(* PLC project CoDeSys External Library Template, WAGO e!COCKPIT e!COCKPIT, author 3S - Smart Software Solutions GmbH *)
(* stored: creationDateTime 2019-10-29T14:38:30.855626, version 3.5.5.30, modificationDateTime 2019-10-29T14:38:06.5373783, organization 3S - Smart Software Solutions GmbH *)
(* Library project template with all possible element types, docu and a sample project structure *)

FUNCTION_BLOCK fbPPPSAnalizatorDirisA40
  VAR_INPUT
    sKomunikat : alSTRINGKomunikat;  (* komunikat z systemu zewnętrznego *)
    intTablicaKomunikatowRozmiar : INT;  (* rozmiar tablicy danych wysyłkowych *)
    xTablicaKomunikatowHold : BOOL;  (* wstrzymanie komunikacji mniej ważnych komunikatów *)
    sIdInstancji : STRING;  (* parametr ID rolety np NS02L*202IBM**** *)
    sIdAplikacji : STRING;  (* parametr ID aplikacji np SO*******ECL*000 *)
    sMnemonik : STRING;  (* mnemonik właściciela - BCB* *)
    sMACAdres : STRING;  (* MAC adres sterownika *)
    sDaneZapasowe : STRING;  (* 6 znaków zapasu *)
    tCzasOpoznieniaRestartu : TIME;  (* czas opóźnienia po którym zaczynają być raportowane wartości *)
    bAdres : BYTE;
    rDeadband : REAL;
    tMinimalnyCzasRaportowania : TIME;
    tMaksymalnyCzasRaportowania : TIME;
    xAutonomizacja : BOOL;
  END_VAR
  VAR_IN_OUT
    arModbusOdczytCykliczny : ARRAY[1..5000] OF typModbusOdczytCykliczny;
    arModbusStatusKomunikacji : ARRAY[1..256] OF INT;
    arTablicaKomunikatow : alARRAYTablicaKomunikatow;
    intTablicaKomunikatowZnacznikZapisu : INT;
  END_VAR
  VAR
    xPierwszySkan : BOOL := TRUE;
    intPetlaPierwszySkan : INT := 1;
    fbTimerBrakuKomunikacji : TON;  (* Kontrola komunikacji urządzenia *)
    xBrakKomunikacjiPLC : BOOL;
    xBrakKomunikacjiIZE : BOOL;
    wNapiecieL1Hi : WORD;  (* Napięcia fazowe *)
    wNapiecieL1Lo : WORD;
    rNapiecieL1 : REAL;
    fbNapiecieL1 : fbFiltrWartoscAnalogowa;
    rNapiecieL1Zaraportowana : REAL;
    rNapiecieL1Pamiec : REAL;
    xBrakZmianyNapiecieL1 : BOOL;
    fbBrakZmianyNapiecieL1Timer : TON;
    xBladBrakZmianyNapiecieL1 : BOOL;
    wNapiecieL2Hi : WORD;
    wNapiecieL2Lo : WORD;
    rNapiecieL2 : REAL;
    fbNapiecieL2 : fbFiltrWartoscAnalogowa;
    rNapiecieL2Zaraportowana : REAL;
    rNapiecieL2Pamiec : REAL;
    xBrakZmianyNapiecieL2 : BOOL;
    fbBrakZmianyNapiecieL2Timer : TON;
    xBladBrakZmianyNapiecieL2 : BOOL;
    wNapiecieL3Hi : WORD;
    wNapiecieL3Lo : WORD;
    rNapiecieL3 : REAL;
    fbNapiecieL3 : fbFiltrWartoscAnalogowa;
    rNapiecieL3Zaraportowana : REAL;
    rNapiecieL3Pamiec : REAL;
    xBrakZmianyNapiecieL3 : BOOL;
    fbBrakZmianyNapiecieL3Timer : TON;
    xBladBrakZmianyNapiecieL3 : BOOL;
    wNapiecieL1L2Hi : WORD;  (* Napięcia przewodowe *)
    wNapiecieL1L2Lo : WORD;
    rNapiecieL1L2 : REAL;
    fbNapiecieL1L2 : fbFiltrWartoscAnalogowa;
    rNapiecieL1L2Zaraportowana : REAL;
    wNapiecieL2L3Hi : WORD;
    wNapiecieL2L3Lo : WORD;
    rNapiecieL2L3 : REAL;
    fbNapiecieL2L3 : fbFiltrWartoscAnalogowa;
    rNapiecieL2L3Zaraportowana : REAL;
    wNapiecieL3L1Hi : WORD;
    wNapiecieL3L1Lo : WORD;
    rNapiecieL3L1 : REAL;
    fbNapiecieL3L1 : fbFiltrWartoscAnalogowa;
    rNapiecieL3L1Zaraportowana : REAL;
    wCzestotliwoscHi : WORD;  (* Częstotliwość *)
    wCzestotliwoscLo : WORD;
    rCzestotliwosc : REAL;
    fbCzestotliwosc : fbFiltrWartoscAnalogowa;
    rCzestotliwoscZaraportowana : REAL;
    wCzasPracyAnalizatoraHi : WORD;  (* Czas pracy *)
    wCzasPracyAnalizatoraLo : WORD;
    rCzasPracyAnalizatora : REAL;
    fbCzasPracyAnalizatora : fbFiltrWartoscAnalogowa;
    rCzasPracyAnalizatoraZaraportowana : REAL;
    wPradL1Hi : WORD;  (* Prądy fazowe *)
    wPradL1Lo : WORD;
    rPradL1 : REAL;
    fbPradL1 : fbFiltrWartoscAnalogowa;
    rPradL1Zaraportowana : REAL;
    rPradL1Pamiec : REAL;
    xBrakZmianyPradL1 : BOOL;
    fbBrakZmianyPradL1Timer : TON;
    xBladBrakZmianyPradL1 : BOOL;
    wPradL2Hi : WORD;
    wPradL2Lo : WORD;
    rPradL2 : REAL;
    fbPradL2 : fbFiltrWartoscAnalogowa;
    rPradL2Zaraportowana : REAL;
    rPradL2Pamiec : REAL;
    xBrakZmianyPradL2 : BOOL;
    fbBrakZmianyPradL2Timer : TON;
    xBladBrakZmianyPradL2 : BOOL;
    wPradL3Hi : WORD;
    wPradL3Lo : WORD;
    rPradL3 : REAL;
    fbPradL3 : fbFiltrWartoscAnalogowa;
    rPradL3Zaraportowana : REAL;
    rPradL3Pamiec : REAL;
    xBrakZmianyPradL3 : BOOL;
    fbBrakZmianyPradL3Timer : TON;
    xBladBrakZmianyPradL3 : BOOL;
    wPradNHi : WORD;
    wPradNLo : WORD;
    rPradN : REAL;
    fbPradN : fbFiltrWartoscAnalogowa;
    rPradNZaraportowana : REAL;
    wPradSredniL1Hi : WORD;  (* Prądy średnie fazowe *)
    wPradSredniL1Lo : WORD;
    rPradSredniL1 : REAL;
    fbPradSredniL1 : fbFiltrWartoscAnalogowa;
    rPradSredniL1Zaraportowana : REAL;
    wPradSredniL2Hi : WORD;
    wPradSredniL2Lo : WORD;
    rPradSredniL2 : REAL;
    fbPradSredniL2 : fbFiltrWartoscAnalogowa;
    rPradSredniL2Zaraportowana : REAL;
    wPradSredniL3Hi : WORD;
    wPradSredniL3Lo : WORD;
    rPradSredniL3 : REAL;
    fbPradSredniL3 : fbFiltrWartoscAnalogowa;
    rPradSredniL3Zaraportowana : REAL;
    rPradSredni : REAL;  (* Prąd średni (I1+I2+I3)/3 *)
    fbPradSredni : fbFiltrWartoscAnalogowa;
    rPradSredniZaraportowana : REAL;
    wMocCzynnaCalkowitaHi : WORD;  (* Moc 3-fazowa czynna *)
    wMocCzynnaCalkowitaLo : WORD;
    rMocCzynnaCalkowita : REAL;
    fbMocCzynnaCalkowita : fbFiltrWartoscAnalogowa;
    rMocCzynnaCalkowitaZaraportowana : REAL;
    wMocBiernaCalkowitaHi : WORD;  (* Moc 3-fazowa bierna *)
    wMocBiernaCalkowitaLo : WORD;
    rMocBiernaCalkowita : REAL;
    fbMocBiernaCalkowita : fbFiltrWartoscAnalogowa;
    rMocBiernaCalkowitaZaraportowana : REAL;
    wMocPozornaCalkowitaHi : WORD;  (* Moc 3-fazowa pozorna *)
    wMocPozornaCalkowitaLo : WORD;
    rMocPozornaCalkowita : REAL;
    fbMocPozornaCalkowita : fbFiltrWartoscAnalogowa;
    rMocPozornaCalkowitaZaraportowana : REAL;
    wWspolczynnikMocyCalkowityHi : WORD;  (* Całkowity współczynnik mocy *)
    wWspolczynnikMocyCalkowityLo : WORD;
    rWspolczynnikMocyCalkowity : REAL;
    fbWspolczynnikMocyCalkowity : fbFiltrWartoscAnalogowa;
    rWspolczynnikMocyCalkowityZaraportowana : REAL;
    wMocCzynnaL1Hi : WORD;  (* Moc Czynna fazowa *)
    wMocCzynnaL1Lo : WORD;
    rMocCzynnaL1 : REAL;
    fbMocCzynnaL1 : fbFiltrWartoscAnalogowa;
    rMocCzynnaL1Zaraportowana : REAL;
    wMocCzynnaL2Hi : WORD;
    wMocCzynnaL2Lo : WORD;
    rMocCzynnaL2 : REAL;
    fbMocCzynnaL2 : fbFiltrWartoscAnalogowa;
    rMocCzynnaL2Zaraportowana : REAL;
    wMocCzynnaL3Hi : WORD;
    wMocCzynnaL3Lo : WORD;
    rMocCzynnaL3 : REAL;
    fbMocCzynnaL3 : fbFiltrWartoscAnalogowa;
    rMocCzynnaL3Zaraportowana : REAL;
    wMocBiernaL1Hi : WORD;  (* Moc Bierna fazowa *)
    wMocBiernaL1Lo : WORD;
    rMocBiernaL1 : REAL;
    fbMocBiernaL1 : fbFiltrWartoscAnalogowa;
    rMocBiernaL1Zaraportowana : REAL;
    wMocBiernaL2Hi : WORD;
    wMocBiernaL2Lo : WORD;
    rMocBiernaL2 : REAL;
    fbMocBiernaL2 : fbFiltrWartoscAnalogowa;
    rMocBiernaL2Zaraportowana : REAL;
    wMocBiernaL3Hi : WORD;
    wMocBiernaL3Lo : WORD;
    rMocBiernaL3 : REAL;
    fbMocBiernaL3 : fbFiltrWartoscAnalogowa;
    rMocBiernaL3Zaraportowana : REAL;
    wMocPozornaL1Hi : WORD;  (* Moc Pozorna fazowa *)
    wMocPozornaL1Lo : WORD;
    rMocPozornaL1 : REAL;
    fbMocPozornaL1 : fbFiltrWartoscAnalogowa;
    rMocPozornaL1Zaraportowana : REAL;
    wMocPozornaL2Hi : WORD;
    wMocPozornaL2Lo : WORD;
    rMocPozornaL2 : REAL;
    fbMocPozornaL2 : fbFiltrWartoscAnalogowa;
    rMocPozornaL2Zaraportowana : REAL;
    wMocPozornaL3Hi : WORD;
    wMocPozornaL3Lo : WORD;
    rMocPozornaL3 : REAL;
    fbMocPozornaL3 : fbFiltrWartoscAnalogowa;
    rMocPozornaL3Zaraportowana : REAL;
    wWspolczynnikMocyL1Hi : WORD;  (* Fazowe współczynniki mocy *)
    wWspolczynnikMocyL1Lo : WORD;
    rWspolczynnikMocyL1 : REAL;
    fbWspolczynnikMocyL1 : fbFiltrWartoscAnalogowa;
    rWspolczynnikMocyL1Zaraportowana : REAL;
    wWspolczynnikMocyL2Hi : WORD;
    wWspolczynnikMocyL2Lo : WORD;
    rWspolczynnikMocyL2 : REAL;
    fbWspolczynnikMocyL2 : fbFiltrWartoscAnalogowa;
    rWspolczynnikMocyL2Zaraportowana : REAL;
    wWspolczynnikMocyL3Hi : WORD;
    wWspolczynnikMocyL3Lo : WORD;
    rWspolczynnikMocyL3 : REAL;
    fbWspolczynnikMocyL3 : fbFiltrWartoscAnalogowa;
    rWspolczynnikMocyL3Zaraportowana : REAL;
    wEnergiaCzynnaPobranaHi : WORD;  (* Energia pobrana *)
    wEnergiaCzynnaPobranaLo : WORD;
    rEnergiaCzynnaPobrana : REAL;
    fbEnergiaCzynnaPobrana : fbFiltrWartoscAnalogowa;
    rEnergiaCzynnaPobranaZaraportowana : REAL;
    wEnergiaBiernaPobranaHi : WORD;
    wEnergiaBiernaPobranaLo : WORD;
    rEnergiaBiernaPobrana : REAL;
    fbEnergiaBiernaPobrana : fbFiltrWartoscAnalogowa;
    rEnergiaBiernaPobranaZaraportowana : REAL;
    wEnergiaPozornaPobranaHi : WORD;
    wEnergiaPozornaPobranaLo : WORD;
    rEnergiaPozornaPobrana : REAL;
    fbEnergiaPozornaPobrana : fbFiltrWartoscAnalogowa;
    rEnergiaPozornaPobranaZaraportowana : REAL;
    wMocCzynnaSredniaHi : WORD;  (* Moc średnia *)
    wMocCzynnaSredniaLo : WORD;
    rMocCzynnaSrednia : REAL;
    fbMocCzynnaSrednia : fbFiltrWartoscAnalogowa;
    rMocCzynnaSredniaZaraportowana : REAL;
    wMocBiernaSredniaHi : WORD;
    wMocBiernaSredniaLo : WORD;
    rMocBiernaSrednia : REAL;
    fbMocBiernaSrednia : fbFiltrWartoscAnalogowa;
    rMocBiernaSredniaZaraportowana : REAL;
    wMocPozornaSredniaHi : WORD;
    wMocPozornaSredniaLo : WORD;
    rMocPozornaSrednia : REAL;
    fbMocPozornaSrednia : fbFiltrWartoscAnalogowa;
    rMocPozornaSredniaZaraportowana : REAL;
    wMaksymalneNapiecieL1Hi : WORD;  (* Maksymalne napięcia fazowe *)
    wMaksymalneNapiecieL1Lo : WORD;
    rMaksymalneNapiecieL1 : REAL;
    fbMaksymalneNapiecieL1 : fbFiltrWartoscAnalogowa;
    rMaksymalneNapiecieL1Zaraportowana : REAL;
    wMaksymalneNapiecieL2Hi : WORD;
    wMaksymalneNapiecieL2Lo : WORD;
    rMaksymalneNapiecieL2 : REAL;
    fbMaksymalneNapiecieL2 : fbFiltrWartoscAnalogowa;
    rMaksymalneNapiecieL2Zaraportowana : REAL;
    wMaksymalneNapiecieL3Hi : WORD;
    wMaksymalneNapiecieL3Lo : WORD;
    rMaksymalneNapiecieL3 : REAL;
    fbMaksymalneNapiecieL3 : fbFiltrWartoscAnalogowa;
    rMaksymalneNapiecieL3Zaraportowana : REAL;
    wTHDNapieciaL1 : WORD;  (* THD napięcia *)
    rTHDNapieciaL1 : REAL;
    fbTHDNapieciaL1 : fbFiltrWartoscAnalogowa;
    rTHDNapieciaL1Zaraportowana : REAL;
    wTHDNapieciaL2 : WORD;
    rTHDNapieciaL2 : REAL;
    fbTHDNapieciaL2 : fbFiltrWartoscAnalogowa;
    rTHDNapieciaL2Zaraportowana : REAL;
    wTHDNapieciaL3 : WORD;
    rTHDNapieciaL3 : REAL;
    fbTHDNapieciaL3 : fbFiltrWartoscAnalogowa;
    rTHDNapieciaL3Zaraportowana : REAL;
    wTHDPraduL1 : WORD;  (* THD prądu *)
    rTHDPraduL1 : REAL;
    fbTHDPraduL1 : fbFiltrWartoscAnalogowa;
    rTHDPraduL1Zaraportowana : REAL;
    wTHDPraduL2 : WORD;
    rTHDPraduL2 : REAL;
    fbTHDPraduL2 : fbFiltrWartoscAnalogowa;
    rTHDPraduL2Zaraportowana : REAL;
    wTHDPraduL3 : WORD;
    rTHDPraduL3 : REAL;
    fbTHDPraduL3 : fbFiltrWartoscAnalogowa;
    rTHDPraduL3Zaraportowana : REAL;
    xPoInicjalizacji : BOOL;  (* inicjalizacja *)
    fbInicjalizacyjnyTimer : TON;
    intStatus : INT := enumPPPSUrzadenieStatus.Prawidlowy;  (* status urządzenia *)
    intStatusZaraportowana : INT;  (* status urządzenia zaraportowany *)
    sDane : alSTRINGKomunikat;
    sWyslanyKomunikat : alSTRINGKomunikat;
    xZadanieRaportu : BOOL;
    sWyslanyKomunikatDummy : alSTRINGKomunikat;
    sKomunikatPamiec : alSTRINGKomunikat;
    intPetla : INT;
    arErrorStan : ARRAY[0..20] OF INT;  (* tablica przechowująca statusy alarmowe *)
    arErrorKlasa : ARRAY[0..20] OF INT;  (* tablica przechowująca klasy danych alarmów *)
    xRaport : BOOL := FALSE;
    xOverFlow : BOOL;
  END_VAR

            (*			
Autor:					Paweł Kąkol, 2018-09-04-PK
Prawa majątkowe: 		Solwena Sp. z o.o., 
Opis:					fb służy do komunikacji po Modbus RTU z analizatorem sieci ECA0 na budynkach PPP Sopot
						Analizator Diris A40
						
Aktualizacje:			2018-11-20-JB: Poprawienie adresów Modbusowych
						2019-01-21-JC: Przeliczanie charakteru mocy biernej oraz współczynnika mocy (czynna/indukcyjna)
						2019-03-26-AWy: Wyłączenie (wykomentowanie) eneregii oddanej czynnej i biernej
						2019-04-01-AWy: Przeliczenie pomocnicze dla mocy czynnej całkowitej
						2019-05-05-AWy: Dodanie bloków włączania autonomizacji i kontroli komunikacji (analogicznie do pozostałych fb). Usunięcie zmiennej xBrakKomunikacji
						2019-08-14-AWy: Przeniesienie xAutonomizacja do VAR_INPUT
						2019-09-04-AWy: Usunięcie bugów z obliczania współczynnika mocy i mocy biernej.
						2019-09-05-Awy: Zmiana sposobu przeliczania wartości odczytanych po modbusie (sklejenie w DINT i konwersja na REAL). Usunięcie energii oddanej czynnej i biernej.
										Zmiana nazwy atrybutu FACTOR na FACTOR3PH.
						2019-10-18-JB: Zmiana dead-bandów.
						2019-10-24-AWy: Zmiana wartości tCzasMinimalny dla czasu pracy analizatora.
	
*)

//inicjalizacja sterownika

fbInicjalizacyjnyTimer(IN := NOT xPoInicjalizacji , PT := tCzasOpoznieniaRestartu);
IF fbInicjalizacyjnyTimer.Q THEN
	rNapiecieL1Zaraportowana := rNapiecieL1;
	rNapiecieL2Zaraportowana := rNapiecieL2;
	rNapiecieL3Zaraportowana :=sdfsdgsdf rNapiecieL3;
	rNapiecieL1L2Zaraportowana := rNapiecieL1L2;
	rNapiecieL2L3Zaraportowana := rNapiecieL2L3;
	rNapiecieL3L1Zaraportowana := rNapiecieL3L1;
	rCzestotliwoscZaraportowana := rCzestotliwosc;
	rCzasPracyAnalizatoraZaraportowana := rCzasPracyAnalizatora;
	rPradL1Zaraportowana := rPradL1;
	rPradL2Zaraportowana := rPradL2;
	rPradL3Zaraportowana := rPradL3;
	rPradNZaraportowana := rPradN;
	rPradSredniL1Zaraportowana := rPradSredniL1;
	rPradSredniL2Zaraportowana := rPradSredniL2;
	rPradSredniL3Zaraportowana := rPradSredniL3;
	rPradSredniZaraportowana := rPradSredni;
	rMocCzynnaCalkowitaZaraportowana := rMocCzynnaCalkowita;
	rMocBiernaCalkowitaZaraportowana := rMocBiernaCalkowita;
	rMocPozornaCalkowitaZaraportowana := rMocPozornaCalkowita;
	rWspolczynnikMocyCalkowityZaraportowana := rWspolczynnikMocyCalkowity;
	rMocCzynnaL1Zaraportowana := rMocCzynnaL1;
	rMocCzynnaL2Zaraportowana := rMocCzynnaL2;
	rMocCzynnaL3Zaraportowana := rMocCzynnaL3;
	rMocBiernaL1Zaraportowana := rMocBiernaL1;
	rMocBiernaL2Zaraportowana := rMocBiernaL2;
	rMocBiernaL3Zaraportowana := rMocBiernaL3;
	rMocPozornaL1Zaraportowana := rMocPozornaL1;
	rMocPozornaL2Zaraportowana := rMocPozornaL2;
	rMocPozornaL3Zaraportowana := rMocPozornaL3;
	rWspolczynnikMocyL1Zaraportowana := rWspolczynnikMocyL1;
	rWspolczynnikMocyL2Zaraportowana := rWspolczynnikMocyL2;
	rWspolczynnikMocyL3Zaraportowana := rWspolczynnikMocyL3;
	rEnergiaCzynnaPobranaZaraportowana := rEnergiaCzynnaPobrana;
	rEnergiaBiernaPobranaZaraportowana := rEnergiaBiernaPobrana;
	rEnergiaPozornaPobranaZaraportowana := rEnergiaPozornaPobrana;
	rMocCzynnaSredniaZaraportowana := rMocCzynnaSrednia;
	rMocBiernaSredniaZaraportowana := rMocBiernaSrednia;
	rMocPozornaSredniaZaraportowana := rMocPozornaSrednia;
	rMaksymalneNapiecieL1Zaraportowana := rMaksymalneNapiecieL1;
	rMaksymalneNapiecieL2Zaraportowana := rMaksymalneNapiecieL2;
	rMaksymalneNapiecieL3Zaraportowana := rMaksymalneNapiecieL3;
	rTHDNapieciaL1Zaraportowana := rTHDNapieciaL1;
	rTHDNapieciaL2Zaraportowana := rTHDNapieciaL2;
	rTHDNapieciaL3Zaraportowana := rTHDNapieciaL3;
	rTHDPraduL1Zaraportowana := rTHDPraduL1;
	rTHDPraduL2Zaraportowana := rTHDPraduL2;
	rTHDPraduL3Zaraportowana := rTHDPraduL3;
	intStatusZaraportowana := intStatus;
	xPoInicjalizacji := TRUE;
	dupa dupa dupa
END_IF

// Włącz autonomizację jeśli sterownik jest w stanie inicjalizacji lub nastąpiło wymuszenie autonomizacji
IF NOT xPoInicjalizacji THEN
	xAutonomizacja := TRUE;
END_IF 

// Kontrola komunikacji
fbTimerBrakuKomunikacji(IN := arModbusStatusKomunikacji[bAdres] = enumModbusStatus.BrakKomunikacji, PT := T#60S);
IF fbTimerBrakuKomunikacji.Q THEN
	xBrakKomunikacjiPLC := TRUE;
ELSE
	xBrakKomunikacjiPLC := FALSE;
END_IF

IF xAutonomizacja THEN
	xBrakKomunikacjiIZE := TRUE;
ELSE
	xBrakKomunikacjiIZE := FALSE;
END_IF

IF xPierwszySkan THEN
	xPierwszySkan := FALSE;
	WHILE arModbusOdczytCykliczny[intPetlaPierwszySkan].bAdresUrzadzenia <> 0 DO
		intPetlaPierwszySkan := intPetlaPierwszySkan + 1;
	END_WHILE

//deklaracja rejestrow do odczytu
	arModbusOdczytCykliczny[intPetlaPierwszySkan].bAdresUrzadzenia := bAdres;
	arModbusOdczytCykliczny[intPetlaPierwszySkan].bFunkcja := TO_BYTE(enumModbusKodyFunkcji.OdczytNRejestrow);
	arModbusOdczytCykliczny[intPetlaPierwszySkan].uiAdresRejestru := 50512;
	arModbusOdczytCykliczny[intPetlaPierwszySkan].ltCzestotliwosc := TIME_TO_LTIME(tMaksymalnyCzasRaportowania);
	arModbusOdczytCykliczny[intPetlaPierwszySkan].pZmiennaReferencyjna := ADR(wCzasPracyAnalizatoraHi);
	intPetlaPierwszySkan := intPetlaPierwszySkan + 1;

	arModbusOdczytCykliczny[intPetlaPierwszySkan].bAdresUrzadzenia := bAdres;
	arModbusOdczytCykliczny[intPetlaPierwszySkan].bFunkcja := TO_BYTE(enumModbusKodyFunkcji.OdczytNRejestrow);
	arModbusOdczytCykliczny[intPetlaPierwszySkan].uiAdresRejestru := 50513;
	arModbusOdczytCykliczny[intPetlaPierwszySkan].ltCzestotliwosc := TIME_TO_LTIME(tMaksymalnyCzasRaportowania);
	arModbusOdczytCykliczny[intPetlaPierwszySkan].pZmiennaReferencyjna := ADR(wCzasPracyAnalizatoraLo);
	intPetlaPierwszySkan := intPetlaPierwszySkan + 1;

	arModbusOdczytCykliczny[intPetlaPierwszySkan].bAdresUrzadzenia := bAdres;
	arModbusOdczytCykliczny[intPetlaPierwszySkan].bFunkcja := TO_BYTE(enumModbusKodyFunkcji.OdczytNRejestrow);
	arModbusOdczytCykliczny[intPetlaPierwszySkan].uiAdresRejestru := 50514;
	arModbusOdczytCykliczny[intPetlaPierwszySkan].ltCzestotliwosc := TIME_TO_LTIME(tMinimalnyCzasRaportowania);
	arModbusOdczytCykliczny[intPetlaPierwszySkan].pZmiennaReferencyjna := ADR(wNapiecieL1L2Hi);
	intPetlaPierwszySkan := intPetlaPierwszySkan + 1;

	arModbusOdczytCykliczny[intPetlaPierwszySkan].bAdresUrzadzenia := bAdres;
	arModbusOdczytCykliczny[intPetlaPierwszySkan].bFunkcja := TO_BYTE(enumModbusKodyFunkcji.OdczytNRejestrow);
	arModbusOdczytCykliczny[intPetlaPierwszySkan].uiAdresRejestru := 50515;
	arModbusOdczytCykliczny[intPetlaPierwszySkan].ltCzestotliwosc := TIME_TO_LTIME(tMinimalnyCzasRaportowania);
	arModbusOdczytCykliczny[intPetlaPierwszySkan].pZmiennaReferencyjna := ADR(wNapiecieL1L2Lo);
	intPetlaPierwszySkan := intPetlaPierwszySkan + 1;

	arModbusOdczytCykliczny[intPetlaPierwszySkan].bAdresUrzadzenia := bAdres;
	arModbusOdczytCykliczny[intPetlaPierwszySkan].bFunkcja := TO_BYTE(enumModbusKodyFunkcji.OdczytNRejestrow);
	arModbusOdczytCykliczny[intPetlaPierwszySkan].uiAdresRejestru := 50516;
	arModbusOdczytCykliczny[intPetlaPierwszySkan].ltCzestotliwosc := TIME_TO_LTIME(tMinimalnyCzasRaportowania);
	arModbusOdczytCykliczny[intPetlaPierwszySkan].pZmiennaReferencyjna := ADR(wNapiecieL2L3Hi);
	intPetlaPierwszySkan := intPetlaPierwszySkan + 1;
	
	arModbusOdczytCykliczny[intPetlaPierwszySkan].bAdresUrzadzenia := bAdres;
	arModbusOdczytCykliczny[intPetlaPierwszySkan].bFunkcja := TO_BYTE(enumModbusKodyFunkcji.OdczytNRejestrow);
	arModbusOdczytCykliczny[intPetlaPierwszySkan].uiAdresRejestru := 50517;
	arModbusOdczytCykliczny[intPetlaPierwszySkan].ltCzestotliwosc := TIME_TO_LTIME(tMinimalnyCzasRaportowania);
	arModbusOdczytCykliczny[intPetlaPierwszySkan].pZmiennaReferencyjna := ADR(wNapiecieL2L3Lo);
	intPetlaPierwszySkan := intPetlaPierwszySkan + 1;

	arModbusOdczytCykliczny[intPetlaPierwszySkan].bAdresUrzadzenia := bAdres;
	arModbusOdczytCykliczny[intPetlaPierwszySkan].bFunkcja := TO_BYTE(enumModbusKodyFunkcji.OdczytNRejestrow);
	arModbusOdczytCykliczny[intPetlaPierwszySkan].uiAdresRejestru := 50518;
	arModbusOdczytCykliczny[intPetlaPierwszySkan].ltCzestotliwosc := TIME_TO_LTIME(tMinimalnyCzasRaportowania);
	arModbusOdczytCykliczny[intPetlaPierwszySkan].pZmiennaReferencyjna := ADR(wNapiecieL3L1Hi);
	intPetlaPierwszySkan := intPetlaPierwszySkan + 1;
	
	arModbusOdczytCykliczny[intPetlaPierwszySkan].bAdresUrzadzenia := bAdres;
	arModbusOdczytCykliczny[intPetlaPierwszySkan].bFunkcja := TO_BYTE(enumModbusKodyFunkcji.OdczytNRejestrow);
	arModbusOdczytCykliczny[intPetlaPierwszySkan].uiAdresRejestru := 50519;
	arModbusOdczytCykliczny[intPetlaPierwszySkan].ltCzestotliwosc := TIME_TO_LTIME(tMinimalnyCzasRaportowania);
	arModbusOdczytCykliczny[intPetlaPierwszySkan].pZmiennaReferencyjna := ADR(wNapiecieL3L1Lo);
	intPetlaPierwszySkan := intPetlaPierwszySkan + 1;

	arModbusOdczytCykliczny[intPetlaPierwszySkan].bAdresUrzadzenia := bAdres;
	arModbusOdczytCykliczny[intPetlaPierwszySkan].bFunkcja := TO_BYTE(enumModbusKodyFunkcji.OdczytNRejestrow);
	arModbusOdczytCykliczny[intPetlaPierwszySkan].uiAdresRejestru := 50520;
	arModbusOdczytCykliczny[intPetlaPierwszySkan].ltCzestotliwosc := TIME_TO_LTIME(tMinimalnyCzasRaportowania);
	arModbusOdczytCykliczny[intPetlaPierwszySkan].pZmiennaReferencyjna := ADR(wNapiecieL1Hi);
	intPetlaPierwszySkan := intPetlaPierwszySkan + 1;

	arModbusOdczytCykliczny[intPetlaPierwszySkan].bAdresUrzadzenia := bAdres;
	arModbusOdczytCykliczny[intPetlaPierwszySkan].bFunkcja := TO_BYTE(enumModbusKodyFunkcji.OdczytNRejestrow);
	arModbusOdczytCykliczny[intPetlaPierwszySkan].uiAdresRejestru := 50521;
	arModbusOdczytCykliczny[intPetlaPierwszySkan].ltCzestotliwosc := TIME_TO_LTIME(tMinimalnyCzasRaportowania);
	arModbusOdczytCykliczny[intPetlaPierwszySkan].pZmiennaReferencyjna := ADR(wNapiecieL1Lo);
	intPetlaPierwszySkan := intPetlaPierwszySkan + 1;

	arModbusOdczytCykliczny[intPetlaPierwszySkan].bAdresUrzadzenia := bAdres;
	arModbusOdczytCykliczny[intPetlaPierwszySkan].bFunkcja := TO_BYTE(enumModbusKodyFunkcji.OdczytNRejestrow);
	arModbusOdczytCykliczny[intPetlaPierwszySkan].uiAdresRejestru := 50522;
	arModbusOdczytCykliczny[intPetlaPierwszySkan].ltCzestotliwosc := TIME_TO_LTIME(tMinimalnyCzasRaportowania);
	arModbusOdczytCykliczny[intPetlaPierwszySkan].pZmiennaReferencyjna := ADR(wNapiecieL2Hi);
	intPetlaPierwszySkan := intPetlaPierwszySkan + 1;
	
	arModbusOdczytCykliczny[intPetlaPierwszySkan].bAdresUrzadzenia := bAdres;
	arModbusOdczytCykliczny[intPetlaPierwszySkan].bFunkcja := TO_BYTE(enumModbusKodyFunkcji.OdczytNRejestrow);
	arModbusOdczytCykliczny[intPetlaPierwszySkan].uiAdresRejestru := 50523;
	arModbusOdczytCykliczny[intPetlaPierwszySkan].ltCzestotliwosc := TIME_TO_LTIME(tMinimalnyCzasRaportowania);
	arModbusOdczytCykliczny[intPetlaPierwszySkan].pZmiennaReferencyjna := ADR(wNapiecieL2Lo);
	intPetlaPierwszySkan := intPetlaPierwszySkan + 1;

	arModbusOdczytCykliczny[intPetlaPierwszySkan].bAdresUrzadzenia := bAdres;
	arModbusOdczytCykliczny[intPetlaPierwszySkan].bFunkcja := TO_BYTE(enumModbusKodyFunkcji.OdczytNRejestrow);
	arModbusOdczytCykliczny[intPetlaPierwszySkan].uiAdresRejestru := 50524;
	arModbusOdczytCykliczny[intPetlaPierwszySkan].ltCzestotliwosc := TIME_TO_LTIME(tMinimalnyCzasRaportowania);
	arModbusOdczytCykliczny[intPetlaPierwszySkan].pZmiennaReferencyjna := ADR(wNapiecieL3Hi);
	intPetlaPierwszySkan := intPetlaPierwszySkan + 1;
	
	arModbusOdczytCykliczny[intPetlaPierwszySkan].bAdresUrzadzenia := bAdres;
	arModbusOdczytCykliczny[intPetlaPierwszySkan].bFunkcja := TO_BYTE(enumModbusKodyFunkcji.OdczytNRejestrow);
	arModbusOdczytCykliczny[intPetlaPierwszySkan].uiAdresRejestru := 50525;
	arModbusOdczytCykliczny[intPetlaPierwszySkan].ltCzestotliwosc := TIME_TO_LTIME(tMinimalnyCzasRaportowania);
	arModbusOdczytCykliczny[intPetlaPierwszySkan].pZmiennaReferencyjna := ADR(wNapiecieL3Lo);
	intPetlaPierwszySkan := intPetlaPierwszySkan + 1;

	arModbusOdczytCykliczny[intPetlaPierwszySkan].bAdresUrzadzenia := bAdres;
	arModbusOdczytCykliczny[intPetlaPierwszySkan].bFunkcja := TO_BYTE(enumModbusKodyFunkcji.OdczytNRejestrow);
	arModbusOdczytCykliczny[intPetlaPierwszySkan].uiAdresRejestru := 50526;
	arModbusOdczytCykliczny[intPetlaPierwszySkan].ltCzestotliwosc := TIME_TO_LTIME(tMinimalnyCzasRaportowania);
	arModbusOdczytCykliczny[intPetlaPierwszySkan].pZmiennaReferencyjna := ADR(wCzestotliwoscHi);
	intPetlaPierwszySkan := intPetlaPierwszySkan + 1;

	arModbusOdczytCykliczny[intPetlaPierwszySkan].bAdresUrzadzenia := bAdres;
	arModbusOdczytCykliczny[intPetlaPierwszySkan].bFunkcja := TO_BYTE(enumModbusKodyFunkcji.OdczytNRejestrow);
	arModbusOdczytCykliczny[intPetlaPierwszySkan].uiAdresRejestru := 50527;
	arModbusOdczytCykliczny[intPetlaPierwszySkan].ltCzestotliwosc := TIME_TO_LTIME(tMinimalnyCzasRaportowania);
	arModbusOdczytCykliczny[intPetlaPierwszySkan].pZmiennaReferencyjna := ADR(wCzestotliwoscLo);
	intPetlaPierwszySkan := intPetlaPierwszySkan + 1;

	arModbusOdczytCykliczny[intPetlaPierwszySkan].bAdresUrzadzenia := bAdres;
	arModbusOdczytCykliczny[intPetlaPierwszySkan].bFunkcja := TO_BYTE(enumModbusKodyFunkcji.OdczytNRejestrow);
	arModbusOdczytCykliczny[intPetlaPierwszySkan].uiAdresRejestru := 50528;
	arModbusOdczytCykliczny[intPetlaPierwszySkan].ltCzestotliwosc := TIME_TO_LTIME(tMinimalnyCzasRaportowania);
	arModbusOdczytCykliczny[intPetlaPierwszySkan].pZmiennaReferencyjna := ADR(wPradL1Hi);
	intPetlaPierwszySkan := intPetlaPierwszySkan + 1;

	arModbusOdczytCykliczny[intPetlaPierwszySkan].bAdresUrzadzenia := bAdres;
	arModbusOdczytCykliczny[intPetlaPierwszySkan].bFunkcja := TO_BYTE(enumModbusKodyFunkcji.OdczytNRejestrow);
	arModbusOdczytCykliczny[intPetlaPierwszySkan].uiAdresRejestru := 50529;
	arModbusOdczytCykliczny[intPetlaPierwszySkan].ltCzestotliwosc := TIME_TO_LTIME(tMinimalnyCzasRaportowania);
	arModbusOdczytCykliczny[intPetlaPierwszySkan].pZmiennaReferencyjna := ADR(wPradL1Lo);
	intPetlaPierwszySkan := intPetlaPierwszySkan + 1;

	arModbusOdczytCykliczny[intPetlaPierwszySkan].bAdresUrzadzenia := bAdres;
	arModbusOdczytCykliczny[intPetlaPierwszySkan].bFunkcja := TO_BYTE(enumModbusKodyFunkcji.OdczytNRejestrow);
	arModbusOdczytCykliczny[intPetlaPierwszySkan].uiAdresRejestru := 50530;
	arModbusOdczytCykliczny[intPetlaPierwszySkan].ltCzestotliwosc := TIME_TO_LTIME(tMinimalnyCzasRaportowania);
	arModbusOdczytCykliczny[intPetlaPierwszySkan].pZmiennaReferencyjna := ADR(wPradL2Hi);
	intPetlaPierwszySkan := intPetlaPierwszySkan + 1;

	arModbusOdczytCykliczny[intPetlaPierwszySkan].bAdresUrzadzenia := bAdres;
	arModbusOdczytCykliczny[intPetlaPierwszySkan].bFunkcja := TO_BYTE(enumModbusKodyFunkcji.OdczytNRejestrow);
	arModbusOdczytCykliczny[intPetlaPierwszySkan].uiAdresRejestru := 50531;
	arModbusOdczytCykliczny[intPetlaPierwszySkan].ltCzestotliwosc := TIME_TO_LTIME(tMinimalnyCzasRaportowania);
	arModbusOdczytCykliczny[intPetlaPierwszySkan].pZmiennaReferencyjna := ADR(wPradL2Lo);
	intPetlaPierwszySkan := intPetlaPierwszySkan + 1;

	arModbusOdczytCykliczny[intPetlaPierwszySkan].bAdresUrzadzenia := bAdres;
	arModbusOdczytCykliczny[intPetlaPierwszySkan].bFunkcja := TO_BYTE(enumModbusKodyFunkcji.OdczytNRejestrow);
	arModbusOdczytCykliczny[intPetlaPierwszySkan].uiAdresRejestru := 50532;
	arModbusOdczytCykliczny[intPetlaPierwszySkan].ltCzestotliwosc := TIME_TO_LTIME(tMinimalnyCzasRaportowania);
	arModbusOdczytCykliczny[intPetlaPierwszySkan].pZmiennaReferencyjna := ADR(wPradL3Hi);
	intPetlaPierwszySkan := intPetlaPierwszySkan + 1;

	arModbusOdczytCykliczny[intPetlaPierwszySkan].bAdresUrzadzenia := bAdres;
	arModbusOdczytCykliczny[intPetlaPierwszySkan].bFunkcja := TO_BYTE(enumModbusKodyFunkcji.OdczytNRejestrow);
	arModbusOdczytCykliczny[intPetlaPierwszySkan].uiAdresRejestru := 50533;
	arModbusOdczytCykliczny[intPetlaPierwszySkan].ltCzestotliwosc := TIME_TO_LTIME(tMinimalnyCzasRaportowania);
	arModbusOdczytCykliczny[intPetlaPierwszySkan].pZmiennaReferencyjna := ADR(wPradL3Lo);
	intPetlaPierwszySkan := intPetlaPierwszySkan + 1;

	arModbusOdczytCykliczny[intPetlaPierwszySkan].bAdresUrzadzenia := bAdres;
	arModbusOdczytCykliczny[intPetlaPierwszySkan].bFunkcja := TO_BYTE(enumModbusKodyFunkcji.OdczytNRejestrow);
	arModbusOdczytCykliczny[intPetlaPierwszySkan].uiAdresRejestru := 50534;
	arModbusOdczytCykliczny[intPetlaPierwszySkan].ltCzestotliwosc := TIME_TO_LTIME(tMinimalnyCzasRaportowania);
	arModbusOdczytCykliczny[intPetlaPierwszySkan].pZmiennaReferencyjna := ADR(wPradNHi);
	intPetlaPierwszySkan := intPetlaPierwszySkan + 1;

	arModbusOdczytCykliczny[intPetlaPierwszySkan].bAdresUrzadzenia := bAdres;
	arModbusOdczytCykliczny[intPetlaPierwszySkan].bFunkcja := TO_BYTE(enumModbusKodyFunkcji.OdczytNRejestrow);
	arModbusOdczytCykliczny[intPetlaPierwszySkan].uiAdresRejestru := 50535;
	arModbusOdczytCykliczny[intPetlaPierwszySkan].ltCzestotliwosc := TIME_TO_LTIME(tMinimalnyCzasRaportowania);
	arModbusOdczytCykliczny[intPetlaPierwszySkan].pZmiennaReferencyjna := ADR(wPradNLo);
	intPetlaPierwszySkan := intPetlaPierwszySkan + 1;
	
	arModbusOdczytCykliczny[intPetlaPierwszySkan].bAdresUrzadzenia := bAdres;
	arModbusOdczytCykliczny[intPetlaPierwszySkan].bFunkcja := TO_BYTE(enumModbusKodyFunkcji.OdczytNRejestrow);
	arModbusOdczytCykliczny[intPetlaPierwszySkan].uiAdresRejestru := 50536;
	arModbusOdczytCykliczny[intPetlaPierwszySkan].ltCzestotliwosc := TIME_TO_LTIME(tMinimalnyCzasRaportowania);
	arModbusOdczytCykliczny[intPetlaPierwszySkan].pZmiennaReferencyjna := ADR(wMocCzynnaCalkowitaHi);
	intPetlaPierwszySkan := intPetlaPierwszySkan + 1;
	
	arModbusOdczytCykliczny[intPetlaPierwszySkan].bAdresUrzadzenia := bAdres;
	arModbusOdczytCykliczny[intPetlaPierwszySkan].bFunkcja := TO_BYTE(enumModbusKodyFunkcji.OdczytNRejestrow);
	arModbusOdczytCykliczny[intPetlaPierwszySkan].uiAdresRejestru := 50537;
	arModbusOdczytCykliczny[intPetlaPierwszySkan].ltCzestotliwosc := TIME_TO_LTIME(tMinimalnyCzasRaportowania);
	arModbusOdczytCykliczny[intPetlaPierwszySkan].pZmiennaReferencyjna := ADR(wMocCzynnaCalkowitaLo);
	intPetlaPierwszySkan := intPetlaPierwszySkan + 1;
	
	arModbusOdczytCykliczny[intPetlaPierwszySkan].bAdresUrzadzenia := bAdres;
	arModbusOdczytCykliczny[intPetlaPierwszySkan].bFunkcja := TO_BYTE(enumModbusKodyFunkcji.OdczytNRejestrow);
	arModbusOdczytCykliczny[intPetlaPierwszySkan].uiAdresRejestru := 50538;
	arModbusOdczytCykliczny[intPetlaPierwszySkan].ltCzestotliwosc := TIME_TO_LTIME(tMinimalnyCzasRaportowania);
	arModbusOdczytCykliczny[intPetlaPierwszySkan].pZmiennaReferencyjna := ADR(wMocBiernaCalkowitaHi);
	intPetlaPierwszySkan := intPetlaPierwszySkan + 1;
	
	arModbusOdczytCykliczny[intPetlaPierwszySkan].bAdresUrzadzenia := bAdres;
	arModbusOdczytCykliczny[intPetlaPierwszySkan].bFunkcja := TO_BYTE(enumModbusKodyFunkcji.OdczytNRejestrow);
	arModbusOdczytCykliczny[intPetlaPierwszySkan].uiAdresRejestru := 50539;
	arModbusOdczytCykliczny[intPetlaPierwszySkan].ltCzestotliwosc := TIME_TO_LTIME(tMinimalnyCzasRaportowania);
	arModbusOdczytCykliczny[intPetlaPierwszySkan].pZmiennaReferencyjna := ADR(wMocBiernaCalkowitaLo);
	intPetlaPierwszySkan := intPetlaPierwszySkan + 1;
	
	arModbusOdczytCykliczny[intPetlaPierwszySkan].bAdresUrzadzenia := bAdres;
	arModbusOdczytCykliczny[intPetlaPierwszySkan].bFunkcja := TO_BYTE(enumModbusKodyFunkcji.OdczytNRejestrow);
	arModbusOdczytCykliczny[intPetlaPierwszySkan].uiAdresRejestru := 50540;
	arModbusOdczytCykliczny[intPetlaPierwszySkan].ltCzestotliwosc := TIME_TO_LTIME(tMinimalnyCzasRaportowania);
	arModbusOdczytCykliczny[intPetlaPierwszySkan].pZmiennaReferencyjna := ADR(wMocPozornaCalkowitaHi);
	intPetlaPierwszySkan := intPetlaPierwszySkan + 1;
	
	arModbusOdczytCykliczny[intPetlaPierwszySkan].bAdresUrzadzenia := bAdres;
	arModbusOdczytCykliczny[intPetlaPierwszySkan].bFunkcja := TO_BYTE(enumModbusKodyFunkcji.OdczytNRejestrow);
	arModbusOdczytCykliczny[intPetlaPierwszySkan].uiAdresRejestru := 50541;
	arModbusOdczytCykliczny[intPetlaPierwszySkan].ltCzestotliwosc := TIME_TO_LTIME(tMinimalnyCzasRaportowania);
	arModbusOdczytCykliczny[intPetlaPierwszySkan].pZmiennaReferencyjna := ADR(wMocPozornaCalkowitaLo);
	intPetlaPierwszySkan := intPetlaPierwszySkan + 1;
	
	arModbusOdczytCykliczny[intPetlaPierwszySkan].bAdresUrzadzenia := bAdres;
	arModbusOdczytCykliczny[intPetlaPierwszySkan].bFunkcja := TO_BYTE(enumModbusKodyFunkcji.OdczytNRejestrow);
	arModbusOdczytCykliczny[intPetlaPierwszySkan].uiAdresRejestru := 50542;
	arModbusOdczytCykliczny[intPetlaPierwszySkan].ltCzestotliwosc := TIME_TO_LTIME(tMinimalnyCzasRaportowania);
	arModbusOdczytCykliczny[intPetlaPierwszySkan].pZmiennaReferencyjna := ADR(wWspolczynnikMocyCalkowityHi);
	intPetlaPierwszySkan := intPetlaPierwszySkan + 1;
	
	arModbusOdczytCykliczny[intPetlaPierwszySkan].bAdresUrzadzenia := bAdres;
	arModbusOdczytCykliczny[intPetlaPierwszySkan].bFunkcja := TO_BYTE(enumModbusKodyFunkcji.OdczytNRejestrow);
	arModbusOdczytCykliczny[intPetlaPierwszySkan].uiAdresRejestru := 50543;
	arModbusOdczytCykliczny[intPetlaPierwszySkan].ltCzestotliwosc := TIME_TO_LTIME(tMinimalnyCzasRaportowania);
	arModbusOdczytCykliczny[intPetlaPierwszySkan].pZmiennaReferencyjna := ADR(wWspolczynnikMocyCalkowityLo);
	intPetlaPierwszySkan := intPetlaPierwszySkan + 1;

	arModbusOdczytCykliczny[intPetlaPierwszySkan].bAdresUrzadzenia := bAdres;
	arModbusOdczytCykliczny[intPetlaPierwszySkan].bFunkcja := TO_BYTE(enumModbusKodyFunkcji.OdczytNRejestrow);
	arModbusOdczytCykliczny[intPetlaPierwszySkan].uiAdresRejestru := 50554;
	arModbusOdczytCykliczny[intPetlaPierwszySkan].ltCzestotliwosc := TIME_TO_LTIME(tMinimalnyCzasRaportowania);
	arModbusOdczytCykliczny[intPetlaPierwszySkan].pZmiennaReferencyjna := ADR(wMocBiernaL3Hi);
	intPetlaPierwszySkan := intPetlaPierwszySkan + 1;

	arModbusOdczytCykliczny[intPetlaPierwszySkan].bAdresUrzadzenia := bAdres;
	arModbusOdczytCykliczny[intPetlaPierwszySkan].bFunkcja := TO_BYTE(enumModbusKodyFunkcji.OdczytNRejestrow);
	arModbusOdczytCykliczny[intPetlaPierwszySkan].uiAdresRejestru := 50555;
	arModbusOdczytCykliczny[intPetlaPierwszySkan].ltCzestotliwosc := TIME_TO_LTIME(tMinimalnyCzasRaportowania);
	arModbusOdczytCykliczny[intPetlaPierwszySkan].pZmiennaReferencyjna := ADR(wMocBiernaL3Lo);
	intPetlaPierwszySkan := intPetlaPierwszySkan + 1;
	
	arModbusOdczytCykliczny[intPetlaPierwszySkan].bAdresUrzadzenia := bAdres;
	arModbusOdczytCykliczny[intPetlaPierwszySkan].bFunkcja := TO_BYTE(enumModbusKodyFunkcji.OdczytNRejestrow);
	arModbusOdczytCykliczny[intPetlaPierwszySkan].uiAdresRejestru := 50552;
	arModbusOdczytCykliczny[intPetlaPierwszySkan].ltCzestotliwosc := TIME_TO_LTIME(tMinimalnyCzasRaportowania);
	arModbusOdczytCykliczny[intPetlaPierwszySkan].pZmiennaReferencyjna := ADR(wMocBiernaL2Hi);
	intPetlaPierwszySkan := intPetlaPierwszySkan + 1;

	arModbusOdczytCykliczny[intPetlaPierwszySkan].bAdresUrzadzenia := bAdres;
	arModbusOdczytCykliczny[intPetlaPierwszySkan].bFunkcja := TO_BYTE(enumModbusKodyFunkcji.OdczytNRejestrow);
	arModbusOdczytCykliczny[intPetlaPierwszySkan].uiAdresRejestru := 50553;
	arModbusOdczytCykliczny[intPetlaPierwszySkan].ltCzestotliwosc := TIME_TO_LTIME(tMinimalnyCzasRaportowania);
	arModbusOdczytCykliczny[intPetlaPierwszySkan].pZmiennaReferencyjna := ADR(wMocBiernaL2Lo);
	intPetlaPierwszySkan := intPetlaPierwszySkan + 1;	
	
	arModbusOdczytCykliczny[intPetlaPierwszySkan].bAdresUrzadzenia := bAdres;
	arModbusOdczytCykliczny[intPetlaPierwszySkan].bFunkcja := TO_BYTE(enumModbusKodyFunkcji.OdczytNRejestrow);
	arModbusOdczytCykliczny[intPetlaPierwszySkan].uiAdresRejestru := 50550;
	arModbusOdczytCykliczny[intPetlaPierwszySkan].ltCzestotliwosc := TIME_TO_LTIME(tMinimalnyCzasRaportowania);
	arModbusOdczytCykliczny[intPetlaPierwszySkan].pZmiennaReferencyjna := ADR(wMocBiernaL1Hi);
	intPetlaPierwszySkan := intPetlaPierwszySkan + 1;

	arModbusOdczytCykliczny[intPetlaPierwszySkan].bAdresUrzadzenia := bAdres;
	arModbusOdczytCykliczny[intPetlaPierwszySkan].bFunkcja := TO_BYTE(enumModbusKodyFunkcji.OdczytNRejestrow);
	arModbusOdczytCykliczny[intPetlaPierwszySkan].uiAdresRejestru := 50551;
	arModbusOdczytCykliczny[intPetlaPierwszySkan].ltCzestotliwosc := TIME_TO_LTIME(tMinimalnyCzasRaportowania);
	arModbusOdczytCykliczny[intPetlaPierwszySkan].pZmiennaReferencyjna := ADR(wMocBiernaL1Lo);
	intPetlaPierwszySkan := intPetlaPierwszySkan + 1;	


	arModbusOdczytCykliczny[intPetlaPierwszySkan].bAdresUrzadzenia := bAdres;
	arModbusOdczytCykliczny[intPetlaPierwszySkan].bFunkcja := TO_BYTE(enumModbusKodyFunkcji.OdczytNRejestrow);
	arModbusOdczytCykliczny[intPetlaPierwszySkan].uiAdresRejestru := 50544;
	arModbusOdczytCykliczny[intPetlaPierwszySkan].ltCzestotliwosc := TIME_TO_LTIME(tMinimalnyCzasRaportowania);
	arModbusOdczytCykliczny[intPetlaPierwszySkan].pZmiennaReferencyjna := ADR(wMocCzynnaL1Hi);
	intPetlaPierwszySkan := intPetlaPierwszySkan + 1;
	
	arModbusOdczytCykliczny[intPetlaPierwszySkan].bAdresUrzadzenia := bAdres;
	arModbusOdczytCykliczny[intPetlaPierwszySkan].bFunkcja := TO_BYTE(enumModbusKodyFunkcji.OdczytNRejestrow);
	arModbusOdczytCykliczny[intPetlaPierwszySkan].uiAdresRejestru := 50545;
	arModbusOdczytCykliczny[intPetlaPierwszySkan].ltCzestotliwosc := TIME_TO_LTIME(tMinimalnyCzasRaportowania);
	arModbusOdczytCykliczny[intPetlaPierwszySkan].pZmiennaReferencyjna := ADR(wMocCzynnaL1Lo);
	intPetlaPierwszySkan := intPetlaPierwszySkan + 1;
	
	arModbusOdczytCykliczny[intPetlaPierwszySkan].bAdresUrzadzenia := bAdres;
	arModbusOdczytCykliczny[intPetlaPierwszySkan].bFunkcja := TO_BYTE(enumModbusKodyFunkcji.OdczytNRejestrow);
	arModbusOdczytCykliczny[intPetlaPierwszySkan].uiAdresRejestru := 50546;
	arModbusOdczytCykliczny[intPetlaPierwszySkan].ltCzestotliwosc := TIME_TO_LTIME(tMinimalnyCzasRaportowania);
	arModbusOdczytCykliczny[intPetlaPierwszySkan].pZmiennaReferencyjna := ADR(wMocCzynnaL2Hi);
	intPetlaPierwszySkan := intPetlaPierwszySkan + 1;
	
	arModbusOdczytCykliczny[intPetlaPierwszySkan].bAdresUrzadzenia := bAdres;
	arModbusOdczytCykliczny[intPetlaPierwszySkan].bFunkcja := TO_BYTE(enumModbusKodyFunkcji.OdczytNRejestrow);
	arModbusOdczytCykliczny[intPetlaPierwszySkan].uiAdresRejestru := 50547;
	arModbusOdczytCykliczny[intPetlaPierwszySkan].ltCzestotliwosc := TIME_TO_LTIME(tMinimalnyCzasRaportowania);
	arModbusOdczytCykliczny[intPetlaPierwszySkan].pZmiennaReferencyjna := ADR(wMocCzynnaL2Lo);
	intPetlaPierwszySkan := intPetlaPierwszySkan + 1;
	
	arModbusOdczytCykliczny[intPetlaPierwszySkan].bAdresUrzadzenia := bAdres;
	arModbusOdczytCykliczny[intPetlaPierwszySkan].bFunkcja := TO_BYTE(enumModbusKodyFunkcji.OdczytNRejestrow);
	arModbusOdczytCykliczny[intPetlaPierwszySkan].uiAdresRejestru := 50548;
	arModbusOdczytCykliczny[intPetlaPierwszySkan].ltCzestotliwosc := TIME_TO_LTIME(tMinimalnyCzasRaportowania);
	arModbusOdczytCykliczny[intPetlaPierwszySkan].pZmiennaReferencyjna := ADR(wMocCzynnaL3Hi);
	intPetlaPierwszySkan := intPetlaPierwszySkan + 1;
	
	arModbusOdczytCykliczny[intPetlaPierwszySkan].bAdresUrzadzenia := bAdres;
	arModbusOdczytCykliczny[intPetlaPierwszySkan].bFunkcja := TO_BYTE(enumModbusKodyFunkcji.OdczytNRejestrow);
	arModbusOdczytCykliczny[intPetlaPierwszySkan].uiAdresRejestru := 50549;
	arModbusOdczytCykliczny[intPetlaPierwszySkan].ltCzestotliwosc := TIME_TO_LTIME(tMinimalnyCzasRaportowania);
	arModbusOdczytCykliczny[intPetlaPierwszySkan].pZmiennaReferencyjna := ADR(wMocCzynnaL3Lo);
	intPetlaPierwszySkan := intPetlaPierwszySkan + 1;	
	
	arModbusOdczytCykliczny[intPetlaPierwszySkan].bAdresUrzadzenia := bAdres;
	arModbusOdczytCykliczny[intPetlaPierwszySkan].bFunkcja := TO_BYTE(enumModbusKodyFunkcji.OdczytNRejestrow);
	arModbusOdczytCykliczny[intPetlaPierwszySkan].uiAdresRejestru := 50556;
	arModbusOdczytCykliczny[intPetlaPierwszySkan].ltCzestotliwosc := TIME_TO_LTIME(tMinimalnyCzasRaportowania);
	arModbusOdczytCykliczny[intPetlaPierwszySkan].pZmiennaReferencyjna := ADR(wMocPozornaL1Hi);
	intPetlaPierwszySkan := intPetlaPierwszySkan + 1;

	arModbusOdczytCykliczny[intPetlaPierwszySkan].bAdresUrzadzenia := bAdres;
	arModbusOdczytCykliczny[intPetlaPierwszySkan].bFunkcja := TO_BYTE(enumModbusKodyFunkcji.OdczytNRejestrow);
	arModbusOdczytCykliczny[intPetlaPierwszySkan].uiAdresRejestru := 50557;
	arModbusOdczytCykliczny[intPetlaPierwszySkan].ltCzestotliwosc := TIME_TO_LTIME(tMinimalnyCzasRaportowania);
	arModbusOdczytCykliczny[intPetlaPierwszySkan].pZmiennaReferencyjna := ADR(wMocPozornaL1Lo);
	intPetlaPierwszySkan := intPetlaPierwszySkan + 1;	

	arModbusOdczytCykliczny[intPetlaPierwszySkan].bAdresUrzadzenia := bAdres;
	arModbusOdczytCykliczny[intPetlaPierwszySkan].bFunkcja := TO_BYTE(enumModbusKodyFunkcji.OdczytNRejestrow);
	arModbusOdczytCykliczny[intPetlaPierwszySkan].uiAdresRejestru := 50558;
	arModbusOdczytCykliczny[intPetlaPierwszySkan].ltCzestotliwosc := TIME_TO_LTIME(tMinimalnyCzasRaportowania);
	arModbusOdczytCykliczny[intPetlaPierwszySkan].pZmiennaReferencyjna := ADR(wMocPozornaL2Hi);
	intPetlaPierwszySkan := intPetlaPierwszySkan + 1;

	arModbusOdczytCykliczny[intPetlaPierwszySkan].bAdresUrzadzenia := bAdres;
	arModbusOdczytCykliczny[intPetlaPierwszySkan].bFunkcja := TO_BYTE(enumModbusKodyFunkcji.OdczytNRejestrow);
	arModbusOdczytCykliczny[intPetlaPierwszySkan].uiAdresRejestru := 50559;
	arModbusOdczytCykliczny[intPetlaPierwszySkan].ltCzestotliwosc := TIME_TO_LTIME(tMinimalnyCzasRaportowania);
	arModbusOdczytCykliczny[intPetlaPierwszySkan].pZmiennaReferencyjna := ADR(wMocPozornaL2Lo);
	intPetlaPierwszySkan := intPetlaPierwszySkan + 1;	

	arModbusOdczytCykliczny[intPetlaPierwszySkan].bAdresUrzadzenia := bAdres;
	arModbusOdczytCykliczny[intPetlaPierwszySkan].bFunkcja := TO_BYTE(enumModbusKodyFunkcji.OdczytNRejestrow);
	arModbusOdczytCykliczny[intPetlaPierwszySkan].uiAdresRejestru := 50560;
	arModbusOdczytCykliczny[intPetlaPierwszySkan].ltCzestotliwosc := TIME_TO_LTIME(tMinimalnyCzasRaportowania);
	arModbusOdczytCykliczny[intPetlaPierwszySkan].pZmiennaReferencyjna := ADR(wMocPozornaL3Hi);
	intPetlaPierwszySkan := intPetlaPierwszySkan + 1;

	arModbusOdczytCykliczny[intPetlaPierwszySkan].bAdresUrzadzenia := bAdres;
	arModbusOdczytCykliczny[intPetlaPierwszySkan].bFunkcja := TO_BYTE(enumModbusKodyFunkcji.OdczytNRejestrow);
	arModbusOdczytCykliczny[intPetlaPierwszySkan].uiAdresRejestru := 50561;
	arModbusOdczytCykliczny[intPetlaPierwszySkan].ltCzestotliwosc := TIME_TO_LTIME(tMinimalnyCzasRaportowania);
	arModbusOdczytCykliczny[intPetlaPierwszySkan].pZmiennaReferencyjna := ADR(wMocPozornaL3Lo);
	intPetlaPierwszySkan := intPetlaPierwszySkan + 1;	
	
	arModbusOdczytCykliczny[intPetlaPierwszySkan].bAdresUrzadzenia := bAdres;
	arModbusOdczytCykliczny[intPetlaPierwszySkan].bFunkcja := TO_BYTE(enumModbusKodyFunkcji.OdczytNRejestrow);
	arModbusOdczytCykliczny[intPetlaPierwszySkan].uiAdresRejestru := 50562;
	arModbusOdczytCykliczny[intPetlaPierwszySkan].ltCzestotliwosc := TIME_TO_LTIME(tMinimalnyCzasRaportowania);
	arModbusOdczytCykliczny[intPetlaPierwszySkan].pZmiennaReferencyjna := ADR(wWspolczynnikMocyL1Hi);
	intPetlaPierwszySkan := intPetlaPierwszySkan + 1;

	arModbusOdczytCykliczny[intPetlaPierwszySkan].bAdresUrzadzenia := bAdres;
	arModbusOdczytCykliczny[intPetlaPierwszySkan].bFunkcja := TO_BYTE(enumModbusKodyFunkcji.OdczytNRejestrow);
	arModbusOdczytCykliczny[intPetlaPierwszySkan].uiAdresRejestru := 50563;
	arModbusOdczytCykliczny[intPetlaPierwszySkan].ltCzestotliwosc := TIME_TO_LTIME(tMinimalnyCzasRaportowania);
	arModbusOdczytCykliczny[intPetlaPierwszySkan].pZmiennaReferencyjna := ADR(wWspolczynnikMocyL1Lo);
	intPetlaPierwszySkan := intPetlaPierwszySkan + 1;
	
	arModbusOdczytCykliczny[intPetlaPierwszySkan].bAdresUrzadzenia := bAdres;
	arModbusOdczytCykliczny[intPetlaPierwszySkan].bFunkcja := TO_BYTE(enumModbusKodyFunkcji.OdczytNRejestrow);
	arModbusOdczytCykliczny[intPetlaPierwszySkan].uiAdresRejestru := 50564;
	arModbusOdczytCykliczny[intPetlaPierwszySkan].ltCzestotliwosc := TIME_TO_LTIME(tMinimalnyCzasRaportowania);
	arModbusOdczytCykliczny[intPetlaPierwszySkan].pZmiennaReferencyjna := ADR(wWspolczynnikMocyL2Hi);
	intPetlaPierwszySkan := intPetlaPierwszySkan + 1;

	arModbusOdczytCykliczny[intPetlaPierwszySkan].bAdresUrzadzenia := bAdres;
	arModbusOdczytCykliczny[intPetlaPierwszySkan].bFunkcja := TO_BYTE(enumModbusKodyFunkcji.OdczytNRejestrow);
	arModbusOdczytCykliczny[intPetlaPierwszySkan].uiAdresRejestru := 50565;
	arModbusOdczytCykliczny[intPetlaPierwszySkan].ltCzestotliwosc := TIME_TO_LTIME(tMinimalnyCzasRaportowania);
	arModbusOdczytCykliczny[intPetlaPierwszySkan].pZmiennaReferencyjna := ADR(wWspolczynnikMocyL2Lo);
	intPetlaPierwszySkan := intPetlaPierwszySkan + 1;
	
	arModbusOdczytCykliczny[intPetlaPierwszySkan].bAdresUrzadzenia := bAdres;
	arModbusOdczytCykliczny[intPetlaPierwszySkan].bFunkcja := TO_BYTE(enumModbusKodyFunkcji.OdczytNRejestrow);
	arModbusOdczytCykliczny[intPetlaPierwszySkan].uiAdresRejestru := 50566;
	arModbusOdczytCykliczny[intPetlaPierwszySkan].ltCzestotliwosc := TIME_TO_LTIME(tMinimalnyCzasRaportowania);
	arModbusOdczytCykliczny[intPetlaPierwszySkan].pZmiennaReferencyjna := ADR(wWspolczynnikMocyL3Hi);
	intPetlaPierwszySkan := intPetlaPierwszySkan + 1;

	arModbusOdczytCykliczny[intPetlaPierwszySkan].bAdresUrzadzenia := bAdres;
	arModbusOdczytCykliczny[intPetlaPierwszySkan].bFunkcja := TO_BYTE(enumModbusKodyFunkcji.OdczytNRejestrow);
	arModbusOdczytCykliczny[intPetlaPierwszySkan].uiAdresRejestru := 50567;
	arModbusOdczytCykliczny[intPetlaPierwszySkan].ltCzestotliwosc := TIME_TO_LTIME(tMinimalnyCzasRaportowania);
	arModbusOdczytCykliczny[intPetlaPierwszySkan].pZmiennaReferencyjna := ADR(wWspolczynnikMocyL3Lo);
	intPetlaPierwszySkan := intPetlaPierwszySkan + 1;
	
	arModbusOdczytCykliczny[intPetlaPierwszySkan].bAdresUrzadzenia := bAdres;
	arModbusOdczytCykliczny[intPetlaPierwszySkan].bFunkcja := TO_BYTE(enumModbusKodyFunkcji.OdczytNRejestrow);
	arModbusOdczytCykliczny[intPetlaPierwszySkan].uiAdresRejestru := 856;
	arModbusOdczytCykliczny[intPetlaPierwszySkan].ltCzestotliwosc := TIME_TO_LTIME(tMinimalnyCzasRaportowania);
	arModbusOdczytCykliczny[intPetlaPierwszySkan].pZmiennaReferencyjna := ADR(wEnergiaCzynnaPobranaHi);
	intPetlaPierwszySkan := intPetlaPierwszySkan + 1;

	arModbusOdczytCykliczny[intPetlaPierwszySkan].bAdresUrzadzenia := bAdres;
	arModbusOdczytCykliczny[intPetlaPierwszySkan].bFunkcja := TO_BYTE(enumModbusKodyFunkcji.OdczytNRejestrow);
	arModbusOdczytCykliczny[intPetlaPierwszySkan].uiAdresRejestru := 857;
	arModbusOdczytCykliczny[intPetlaPierwszySkan].ltCzestotliwosc := TIME_TO_LTIME(tMinimalnyCzasRaportowania);
	arModbusOdczytCykliczny[intPetlaPierwszySkan].pZmiennaReferencyjna := ADR(wEnergiaCzynnaPobranaLo);
	intPetlaPierwszySkan := intPetlaPierwszySkan + 1;
	
	arModbusOdczytCykliczny[intPetlaPierwszySkan].bAdresUrzadzenia := bAdres;
	arModbusOdczytCykliczny[intPetlaPierwszySkan].bFunkcja := TO_BYTE(enumModbusKodyFunkcji.OdczytNRejestrow);
	arModbusOdczytCykliczny[intPetlaPierwszySkan].uiAdresRejestru := 858;
	arModbusOdczytCykliczny[intPetlaPierwszySkan].ltCzestotliwosc := TIME_TO_LTIME(tMinimalnyCzasRaportowania);
	arModbusOdczytCykliczny[intPetlaPierwszySkan].pZmiennaReferencyjna := ADR(wEnergiaBiernaPobranaHi);
	intPetlaPierwszySkan := intPetlaPierwszySkan + 1;

	arModbusOdczytCykliczny[intPetlaPierwszySkan].bAdresUrzadzenia := bAdres;
	arModbusOdczytCykliczny[intPetlaPierwszySkan].bFunkcja := TO_BYTE(enumModbusKodyFunkcji.OdczytNRejestrow);
	arModbusOdczytCykliczny[intPetlaPierwszySkan].uiAdresRejestru := 859;
	arModbusOdczytCykliczny[intPetlaPierwszySkan].ltCzestotliwosc := TIME_TO_LTIME(tMinimalnyCzasRaportowania);
	arModbusOdczytCykliczny[intPetlaPierwszySkan].pZmiennaReferencyjna := ADR(wEnergiaBiernaPobranaLo);
	intPetlaPierwszySkan := intPetlaPierwszySkan + 1;
	
	arModbusOdczytCykliczny[intPetlaPierwszySkan].bAdresUrzadzenia := bAdres;
	arModbusOdczytCykliczny[intPetlaPierwszySkan].bFunkcja := TO_BYTE(enumModbusKodyFunkcji.OdczytNRejestrow);
	arModbusOdczytCykliczny[intPetlaPierwszySkan].uiAdresRejestru := 860;
	arModbusOdczytCykliczny[intPetlaPierwszySkan].ltCzestotliwosc := TIME_TO_LTIME(tMinimalnyCzasRaportowania);
	arModbusOdczytCykliczny[intPetlaPierwszySkan].pZmiennaReferencyjna := ADR(wEnergiaPozornaPobranaHi);
	intPetlaPierwszySkan := intPetlaPierwszySkan + 1;

	arModbusOdczytCykliczny[intPetlaPierwszySkan].bAdresUrzadzenia := bAdres;
	arModbusOdczytCykliczny[intPetlaPierwszySkan].bFunkcja := TO_BYTE(enumModbusKodyFunkcji.OdczytNRejestrow);
	arModbusOdczytCykliczny[intPetlaPierwszySkan].uiAdresRejestru := 861;
	arModbusOdczytCykliczny[intPetlaPierwszySkan].ltCzestotliwosc := TIME_TO_LTIME(tMinimalnyCzasRaportowania);
	arModbusOdczytCykliczny[intPetlaPierwszySkan].pZmiennaReferencyjna := ADR(wEnergiaPozornaPobranaLo);
	intPetlaPierwszySkan := intPetlaPierwszySkan + 1;
	
	arModbusOdczytCykliczny[intPetlaPierwszySkan].bAdresUrzadzenia := bAdres;
	arModbusOdczytCykliczny[intPetlaPierwszySkan].bFunkcja := TO_BYTE(enumModbusKodyFunkcji.OdczytNRejestrow);
	arModbusOdczytCykliczny[intPetlaPierwszySkan].uiAdresRejestru := 51038;
	arModbusOdczytCykliczny[intPetlaPierwszySkan].ltCzestotliwosc := TIME_TO_LTIME(tMinimalnyCzasRaportowania);
	arModbusOdczytCykliczny[intPetlaPierwszySkan].pZmiennaReferencyjna := ADR(wPradSredniL1Hi);
	intPetlaPierwszySkan := intPetlaPierwszySkan + 1;

	arModbusOdczytCykliczny[intPetlaPierwszySkan].bAdresUrzadzenia := bAdres;
	arModbusOdczytCykliczny[intPetlaPierwszySkan].bFunkcja := TO_BYTE(enumModbusKodyFunkcji.OdczytNRejestrow);
	arModbusOdczytCykliczny[intPetlaPierwszySkan].uiAdresRejestru := 51039;
	arModbusOdczytCykliczny[intPetlaPierwszySkan].ltCzestotliwosc := TIME_TO_LTIME(tMinimalnyCzasRaportowania);
	arModbusOdczytCykliczny[intPetlaPierwszySkan].pZmiennaReferencyjna := ADR(wPradSredniL1Lo);
	intPetlaPierwszySkan := intPetlaPierwszySkan + 1;
	
	arModbusOdczytCykliczny[intPetlaPierwszySkan].bAdresUrzadzenia := bAdres;
	arModbusOdczytCykliczny[intPetlaPierwszySkan].bFunkcja := TO_BYTE(enumModbusKodyFunkcji.OdczytNRejestrow);
	arModbusOdczytCykliczny[intPetlaPierwszySkan].uiAdresRejestru := 51040;
	arModbusOdczytCykliczny[intPetlaPierwszySkan].ltCzestotliwosc := TIME_TO_LTIME(tMinimalnyCzasRaportowania);
	arModbusOdczytCykliczny[intPetlaPierwszySkan].pZmiennaReferencyjna := ADR(wPradSredniL2Hi);
	intPetlaPierwszySkan := intPetlaPierwszySkan + 1;

	arModbusOdczytCykliczny[intPetlaPierwszySkan].bAdresUrzadzenia := bAdres;
	arModbusOdczytCykliczny[intPetlaPierwszySkan].bFunkcja := TO_BYTE(enumModbusKodyFunkcji.OdczytNRejestrow);
	arModbusOdczytCykliczny[intPetlaPierwszySkan].uiAdresRejestru := 51041;
	arModbusOdczytCykliczny[intPetlaPierwszySkan].ltCzestotliwosc := TIME_TO_LTIME(tMinimalnyCzasRaportowania);
	arModbusOdczytCykliczny[intPetlaPierwszySkan].pZmiennaReferencyjna := ADR(wPradSredniL2Lo);
	intPetlaPierwszySkan := intPetlaPierwszySkan + 1;
	
	arModbusOdczytCykliczny[intPetlaPierwszySkan].bAdresUrzadzenia := bAdres;
	arModbusOdczytCykliczny[intPetlaPierwszySkan].bFunkcja := TO_BYTE(enumModbusKodyFunkcji.OdczytNRejestrow);
	arModbusOdczytCykliczny[intPetlaPierwszySkan].uiAdresRejestru := 51042;
	arModbusOdczytCykliczny[intPetlaPierwszySkan].ltCzestotliwosc := TIME_TO_LTIME(tMinimalnyCzasRaportowania);
	arModbusOdczytCykliczny[intPetlaPierwszySkan].pZmiennaReferencyjna := ADR(wPradSredniL3Hi);
	intPetlaPierwszySkan := intPetlaPierwszySkan + 1;

	arModbusOdczytCykliczny[intPetlaPierwszySkan].bAdresUrzadzenia := bAdres;
	arModbusOdczytCykliczny[intPetlaPierwszySkan].bFunkcja := TO_BYTE(enumModbusKodyFunkcji.OdczytNRejestrow);
	arModbusOdczytCykliczny[intPetlaPierwszySkan].uiAdresRejestru := 51043;
	arModbusOdczytCykliczny[intPetlaPierwszySkan].ltCzestotliwosc := TIME_TO_LTIME(tMinimalnyCzasRaportowania);
	arModbusOdczytCykliczny[intPetlaPierwszySkan].pZmiennaReferencyjna := ADR(wPradSredniL3Lo);
	intPetlaPierwszySkan := intPetlaPierwszySkan + 1;

	arModbusOdczytCykliczny[intPetlaPierwszySkan].bAdresUrzadzenia := bAdres;
	arModbusOdczytCykliczny[intPetlaPierwszySkan].bFunkcja := TO_BYTE(enumModbusKodyFunkcji.OdczytNRejestrow);
	arModbusOdczytCykliczny[intPetlaPierwszySkan].uiAdresRejestru := 51046;
	arModbusOdczytCykliczny[intPetlaPierwszySkan].ltCzestotliwosc := TIME_TO_LTIME(tMinimalnyCzasRaportowania);
	arModbusOdczytCykliczny[intPetlaPierwszySkan].pZmiennaReferencyjna := ADR(wMocCzynnaSredniaHi);
	intPetlaPierwszySkan := intPetlaPierwszySkan + 1;

	arModbusOdczytCykliczny[intPetlaPierwszySkan].bAdresUrzadzenia := bAdres;
	arModbusOdczytCykliczny[intPetlaPierwszySkan].bFunkcja := TO_BYTE(enumModbusKodyFunkcji.OdczytNRejestrow);
	arModbusOdczytCykliczny[intPetlaPierwszySkan].uiAdresRejestru := 51047;
	arModbusOdczytCykliczny[intPetlaPierwszySkan].ltCzestotliwosc := TIME_TO_LTIME(tMinimalnyCzasRaportowania);
	arModbusOdczytCykliczny[intPetlaPierwszySkan].pZmiennaReferencyjna := ADR(wMocCzynnaSredniaLo);
	intPetlaPierwszySkan := intPetlaPierwszySkan + 1;

	arModbusOdczytCykliczny[intPetlaPierwszySkan].bAdresUrzadzenia := bAdres;
	arModbusOdczytCykliczny[intPetlaPierwszySkan].bFunkcja := TO_BYTE(enumModbusKodyFunkcji.OdczytNRejestrow);
	arModbusOdczytCykliczny[intPetlaPierwszySkan].uiAdresRejestru := 51052;
	arModbusOdczytCykliczny[intPetlaPierwszySkan].ltCzestotliwosc := TIME_TO_LTIME(tMinimalnyCzasRaportowania);
	arModbusOdczytCykliczny[intPetlaPierwszySkan].pZmiennaReferencyjna := ADR(wMocBiernaSredniaHi);
	intPetlaPierwszySkan := intPetlaPierwszySkan + 1;

	arModbusOdczytCykliczny[intPetlaPierwszySkan].bAdresUrzadzenia := bAdres;
	arModbusOdczytCykliczny[intPetlaPierwszySkan].bFunkcja := TO_BYTE(enumModbusKodyFunkcji.OdczytNRejestrow);
	arModbusOdczytCykliczny[intPetlaPierwszySkan].uiAdresRejestru := 51053;
	arModbusOdczytCykliczny[intPetlaPierwszySkan].ltCzestotliwosc := TIME_TO_LTIME(tMinimalnyCzasRaportowania);
	arModbusOdczytCykliczny[intPetlaPierwszySkan].pZmiennaReferencyjna := ADR(wMocBiernaSredniaLo);
	intPetlaPierwszySkan := intPetlaPierwszySkan + 1;

	arModbusOdczytCykliczny[intPetlaPierwszySkan].bAdresUrzadzenia := bAdres;
	arModbusOdczytCykliczny[intPetlaPierwszySkan].bFunkcja := TO_BYTE(enumModbusKodyFunkcji.OdczytNRejestrow);
	arModbusOdczytCykliczny[intPetlaPierwszySkan].uiAdresRejestru := 51054;
	arModbusOdczytCykliczny[intPetlaPierwszySkan].ltCzestotliwosc := TIME_TO_LTIME(tMinimalnyCzasRaportowania);
	arModbusOdczytCykliczny[intPetlaPierwszySkan].pZmiennaReferencyjna := ADR(wMocPozornaSredniaHi);
	intPetlaPierwszySkan := intPetlaPierwszySkan + 1;

	arModbusOdczytCykliczny[intPetlaPierwszySkan].bAdresUrzadzenia := bAdres;
	arModbusOdczytCykliczny[intPetlaPierwszySkan].bFunkcja := TO_BYTE(enumModbusKodyFunkcji.OdczytNRejestrow);
	arModbusOdczytCykliczny[intPetlaPierwszySkan].uiAdresRejestru := 51055;
	arModbusOdczytCykliczny[intPetlaPierwszySkan].ltCzestotliwosc := TIME_TO_LTIME(tMinimalnyCzasRaportowania);
	arModbusOdczytCykliczny[intPetlaPierwszySkan].pZmiennaReferencyjna := ADR(wMocPozornaSredniaLo);
	intPetlaPierwszySkan := intPetlaPierwszySkan + 1;

	arModbusOdczytCykliczny[intPetlaPierwszySkan].bAdresUrzadzenia := bAdres;
	arModbusOdczytCykliczny[intPetlaPierwszySkan].bFunkcja := TO_BYTE(enumModbusKodyFunkcji.OdczytNRejestrow);
	arModbusOdczytCykliczny[intPetlaPierwszySkan].uiAdresRejestru := 51062;
	arModbusOdczytCykliczny[intPetlaPierwszySkan].ltCzestotliwosc := TIME_TO_LTIME(tMinimalnyCzasRaportowania);
	arModbusOdczytCykliczny[intPetlaPierwszySkan].pZmiennaReferencyjna := ADR(wMaksymalneNapiecieL1Hi);
	intPetlaPierwszySkan := intPetlaPierwszySkan + 1;

	arModbusOdczytCykliczny[intPetlaPierwszySkan].bAdresUrzadzenia := bAdres;
	arModbusOdczytCykliczny[intPetlaPierwszySkan].bFunkcja := TO_BYTE(enumModbusKodyFunkcji.OdczytNRejestrow);
	arModbusOdczytCykliczny[intPetlaPierwszySkan].uiAdresRejestru := 51063;
	arModbusOdczytCykliczny[intPetlaPierwszySkan].ltCzestotliwosc := TIME_TO_LTIME(tMinimalnyCzasRaportowania);
	arModbusOdczytCykliczny[intPetlaPierwszySkan].pZmiennaReferencyjna := ADR(wMaksymalneNapiecieL1Lo);
	intPetlaPierwszySkan := intPetlaPierwszySkan + 1;

	arModbusOdczytCykliczny[intPetlaPierwszySkan].bAdresUrzadzenia := bAdres;
	arModbusOdczytCykliczny[intPetlaPierwszySkan].bFunkcja := TO_BYTE(enumModbusKodyFunkcji.OdczytNRejestrow);
	arModbusOdczytCykliczny[intPetlaPierwszySkan].uiAdresRejestru := 51064;
	arModbusOdczytCykliczny[intPetlaPierwszySkan].ltCzestotliwosc := TIME_TO_LTIME(tMinimalnyCzasRaportowania);
	arModbusOdczytCykliczny[intPetlaPierwszySkan].pZmiennaReferencyjna := ADR(wMaksymalneNapiecieL2Hi);
	intPetlaPierwszySkan := intPetlaPierwszySkan + 1;

	arModbusOdczytCykliczny[intPetlaPierwszySkan].bAdresUrzadzenia := bAdres;
	arModbusOdczytCykliczny[intPetlaPierwszySkan].bFunkcja := TO_BYTE(enumModbusKodyFunkcji.OdczytNRejestrow);
	arModbusOdczytCykliczny[intPetlaPierwszySkan].uiAdresRejestru := 51065;
	arModbusOdczytCykliczny[intPetlaPierwszySkan].ltCzestotliwosc := TIME_TO_LTIME(tMinimalnyCzasRaportowania);
	arModbusOdczytCykliczny[intPetlaPierwszySkan].pZmiennaReferencyjna := ADR(wMaksymalneNapiecieL2Lo);
	intPetlaPierwszySkan := intPetlaPierwszySkan + 1;

	arModbusOdczytCykliczny[intPetlaPierwszySkan].bAdresUrzadzenia := bAdres;
	arModbusOdczytCykliczny[intPetlaPierwszySkan].bFunkcja := TO_BYTE(enumModbusKodyFunkcji.OdczytNRejestrow);
	arModbusOdczytCykliczny[intPetlaPierwszySkan].uiAdresRejestru := 51066;
	arModbusOdczytCykliczny[intPetlaPierwszySkan].ltCzestotliwosc := TIME_TO_LTIME(tMinimalnyCzasRaportowania);
	arModbusOdczytCykliczny[intPetlaPierwszySkan].pZmiennaReferencyjna := ADR(wMaksymalneNapiecieL3Hi);
	intPetlaPierwszySkan := intPetlaPierwszySkan + 1;

	arModbusOdczytCykliczny[intPetlaPierwszySkan].bAdresUrzadzenia := bAdres;
	arModbusOdczytCykliczny[intPetlaPierwszySkan].bFunkcja := TO_BYTE(enumModbusKodyFunkcji.OdczytNRejestrow);
	arModbusOdczytCykliczny[intPetlaPierwszySkan].uiAdresRejestru := 51067;
	arModbusOdczytCykliczny[intPetlaPierwszySkan].ltCzestotliwosc := TIME_TO_LTIME(tMinimalnyCzasRaportowania);
	arModbusOdczytCykliczny[intPetlaPierwszySkan].pZmiennaReferencyjna := ADR(wMaksymalneNapiecieL3Lo);
	intPetlaPierwszySkan := intPetlaPierwszySkan + 1;

	arModbusOdczytCykliczny[intPetlaPierwszySkan].bAdresUrzadzenia := bAdres;
	arModbusOdczytCykliczny[intPetlaPierwszySkan].bFunkcja := TO_BYTE(enumModbusKodyFunkcji.OdczytNRejestrow);
	arModbusOdczytCykliczny[intPetlaPierwszySkan].uiAdresRejestru := 51539;
	arModbusOdczytCykliczny[intPetlaPierwszySkan].ltCzestotliwosc := TIME_TO_LTIME(tMinimalnyCzasRaportowania);
	arModbusOdczytCykliczny[intPetlaPierwszySkan].pZmiennaReferencyjna := ADR(wTHDNapieciaL1);
	intPetlaPierwszySkan := intPetlaPierwszySkan + 1;

	arModbusOdczytCykliczny[intPetlaPierwszySkan].bAdresUrzadzenia := bAdres;
	arModbusOdczytCykliczny[intPetlaPierwszySkan].bFunkcja := TO_BYTE(enumModbusKodyFunkcji.OdczytNRejestrow);
	arModbusOdczytCykliczny[intPetlaPierwszySkan].uiAdresRejestru := 51540;
	arModbusOdczytCykliczny[intPetlaPierwszySkan].ltCzestotliwosc := TIME_TO_LTIME(tMinimalnyCzasRaportowania);
	arModbusOdczytCykliczny[intPetlaPierwszySkan].pZmiennaReferencyjna := ADR(wTHDNapieciaL2);
	intPetlaPierwszySkan := intPetlaPierwszySkan + 1;

	arModbusOdczytCykliczny[intPetlaPierwszySkan].bAdresUrzadzenia := bAdres;
	arModbusOdczytCykliczny[intPetlaPierwszySkan].bFunkcja := TO_BYTE(enumModbusKodyFunkcji.OdczytNRejestrow);
	arModbusOdczytCykliczny[intPetlaPierwszySkan].uiAdresRejestru := 51541;
	arModbusOdczytCykliczny[intPetlaPierwszySkan].ltCzestotliwosc := TIME_TO_LTIME(tMinimalnyCzasRaportowania);
	arModbusOdczytCykliczny[intPetlaPierwszySkan].pZmiennaReferencyjna := ADR(wTHDNapieciaL3);
	intPetlaPierwszySkan := intPetlaPierwszySkan + 1;

	arModbusOdczytCykliczny[intPetlaPierwszySkan].bAdresUrzadzenia := bAdres;
	arModbusOdczytCykliczny[intPetlaPierwszySkan].bFunkcja := TO_BYTE(enumModbusKodyFunkcji.OdczytNRejestrow);
	arModbusOdczytCykliczny[intPetlaPierwszySkan].uiAdresRejestru := 51542;
	arModbusOdczytCykliczny[intPetlaPierwszySkan].ltCzestotliwosc := TIME_TO_LTIME(tMinimalnyCzasRaportowania);
	arModbusOdczytCykliczny[intPetlaPierwszySkan].pZmiennaReferencyjna := ADR(wTHDPraduL1);
	intPetlaPierwszySkan := intPetlaPierwszySkan + 1;

	arModbusOdczytCykliczny[intPetlaPierwszySkan].bAdresUrzadzenia := bAdres;
	arModbusOdczytCykliczny[intPetlaPierwszySkan].bFunkcja := TO_BYTE(enumModbusKodyFunkcji.OdczytNRejestrow);
	arModbusOdczytCykliczny[intPetlaPierwszySkan].uiAdresRejestru := 51543;
	arModbusOdczytCykliczny[intPetlaPierwszySkan].ltCzestotliwosc := TIME_TO_LTIME(tMinimalnyCzasRaportowania);
	arModbusOdczytCykliczny[intPetlaPierwszySkan].pZmiennaReferencyjna := ADR(wTHDPraduL2);
	intPetlaPierwszySkan := intPetlaPierwszySkan + 1;

	arModbusOdczytCykliczny[intPetlaPierwszySkan].bAdresUrzadzenia := bAdres;
	arModbusOdczytCykliczny[intPetlaPierwszySkan].bFunkcja := TO_BYTE(enumModbusKodyFunkcji.OdczytNRejestrow);
	arModbusOdczytCykliczny[intPetlaPierwszySkan].uiAdresRejestru := 51544;
	arModbusOdczytCykliczny[intPetlaPierwszySkan].ltCzestotliwosc := TIME_TO_LTIME(tMinimalnyCzasRaportowania);
	arModbusOdczytCykliczny[intPetlaPierwszySkan].pZmiennaReferencyjna := ADR(wTHDPraduL3);
	intPetlaPierwszySkan := intPetlaPierwszySkan + 1;
END_IF

//obsluga komunikatu przychodzacego z IZE

